DATA_BLOCK "Conveyor_DB"
{ S7_Optimized_Access := 'TRUE' }
VERSION : 0.1
NON_RETAIN
"FB_Conveyor"

BEGIN

END_DATA_BLOCK
